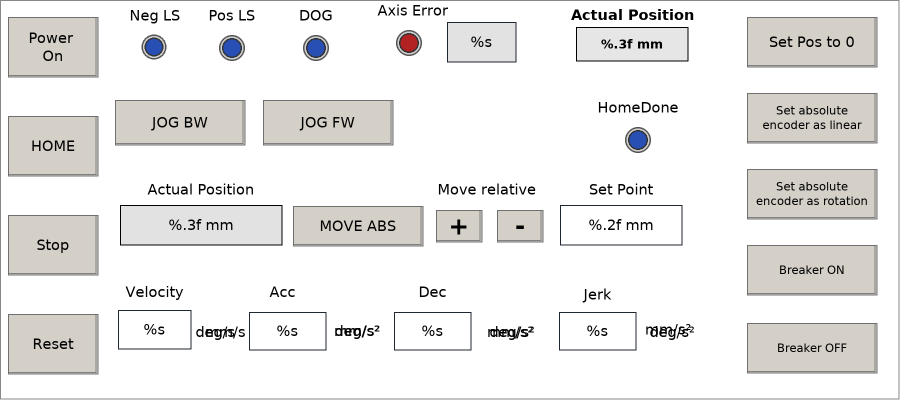
VISUALIZATION AxisHMI_Ex  // 900x400
VAR_IN_OUT
	stAxisHMI	: ST_MotionAxis_MC	;
	mcAxis		: FB_MotionAxis_MC;
	//sAxisName	: STRING			;// Axis Name
	//iAxisID		: INT			;// Axis Id
	xError		: BOOL				;// Axis error flag
END_VAR
    Button (115,100 130x45), "JOG BW", colour toggle: stAxisHMI.mcJog.JogBackwards
        OnMouseDown: execute { stAxisHMI.mcJog.JogBackwards := TRUE; }
        OnMouseUp: execute { stAxisHMI.mcJog.JogBackwards := FALSE; }
    Button (263,100 130x45), "JOG FW", colour toggle: stAxisHMI.mcJog.JogForward
        OnMouseDown: execute { stAxisHMI.mcJog.JogForward := TRUE; }
        OnMouseUp: execute { stAxisHMI.mcJog.JogForward := FALSE; }
    Rectangle (120,205 162x40), "%.3f mm", text variable: stAxisHMI.rActualPosHMI
        OnMouseClick: write the text variable via Default
    Label (141,177 120x25), "Actual Position"
    Button (8,17 90x60), "Power On", colour toggle: stAxisHMI.mcPower.Enable, pressed state: stAxisHMI.mcPower.Enable
        OnMouseClick: toggle stAxisHMI.mcPower.Enable
    Button (8,215 90x60), "Stop", colour toggle: stAxisHMI.mcStop.Execute, invisible if: NOT stAxisHMI.bStopButtonShow
        OnMouseDown: execute { stAxisHMI.mcStop.Execute := TRUE; }
        OnMouseUp: execute { stAxisHMI.mcStop.Execute := FALSE; }
    Button (8,314 90x60), "Reset", colour toggle: stAxisHMI.mcReset.Execute
        OnMouseDown: execute { stAxisHMI.mcReset.Execute := TRUE; }
        OnMouseUp: execute { stAxisHMI.mcReset.Execute := FALSE; }
    Label (111,277 87x30), "Velocity"
    Rectangle (118,310 73x39), "%s", text variable: stAxisHMI.rVeloPers
        OnMouseClick: write the text variable via Default, min 1, max stAxisHMI.rMaxVelocity
    Label (230,277 105x30), "Acc"
    Rectangle (249,312 77x38), "%s", text variable: stAxisHMI.rAcceleration
        OnMouseClick: write stAxisHMI.rAccPers via Default, min 1, max stAxisHMI.rMaxAcceleration
    Lamp1 (139,33 30x28), variable: stAxisHMI.bNegSen, invisible if: NOT stAxisHMI.bNegSensorShow, style: Lamp-Lamp1-Blue
    Label (364,-2 102x25), "Axis Error"
    Rectangle (447,22 69x40), "%s", text variable: stAxisHMI.mcReadStatus.ErrorID
    Lamp1 (394,28 30x30), variable: xError, style: Lamp-Lamp1-Red
    Lamp1 (217,33 30x30), variable: stAxisHMI.bPosSen, invisible if: NOT stAxisHMI.bPosSensorShow, style: Lamp-Lamp1-Blue
    Label (188,3 88x25), "Pos LS", invisible if: NOT stAxisHMI.bPosSensorShow
    Label (111,3 88x25), "Neg LS", invisible if: NOT stAxisHMI.bNegSensorShow
    Rectangle (560,205 122x40), "%.2f mm", text variable: stAxisHMI.rDistance
        OnMouseClick: write the text variable via Default, min 0, max stAxisHMI.rMaxDistance
    Button (293,206 130x40), "MOVE ABS", colour toggle: stAxisHMI.mcMoveAbsolute.Busy, pressed state: stAxisHMI.mcMoveAbsolute.Busy
        OnMouseDown: execute { stAxisHMI.bMoveAbsHMI := TRUE; }
        OnMouseUp: execute { stAxisHMI.bMoveAbsHMI := FALSE; }
    Label (561,177 120x25), "Set Point"
    Button (436,210 46x32), "+", colour toggle: stAxisHMI.mcMoveRelative.Busy, pressed state: stAxisHMI.mcMoveRelative.Busy
        OnMouseDown: execute { stAxisHMI.rPosition := stAxisHMI.rDistance; stAxisHMI.mcMoveRelative.Execute := TRUE; }
        OnMouseUp: execute { stAxisHMI.mcMoveRelative.Execute := FALSE; }
    Button (497,210 46x32), "-", colour toggle: stAxisHMI.mcMoveRelative.Busy, pressed state: stAxisHMI.mcMoveRelative.Busy
        OnMouseDown: execute { stAxisHMI.rPosition := -(stAxisHMI.rDistance); stAxisHMI.mcMoveRelative.Execute := TRUE; }
        OnMouseUp: execute { stAxisHMI.mcMoveRelative.Execute := FALSE; }
    Label (427,177 120x25), "Move relative"
    Label (330,316 55x30), "mm/s²"
    Label (196,317 59x30), "mm/s"
    Label (191,317 49x30), "deg/s", invisible if: NOT stAxisHMI.bUnitDegShow
    Label (328,316 59x30), "deg/s²", invisible if: NOT stAxisHMI.bUnitDegShow
    Label (380,277 105x30), "Dec"
    Rectangle (394,312 77x38), "%s", text variable: stAxisHMI.rDeceleration
        OnMouseClick: write stAxisHMI.rDecPers via Default, min 1, max stAxisHMI.rMaxDeceleration
    Label (483,317 55x30), "mm/s²"
    Label (483,317 59x30), "deg/s²", invisible if: NOT stAxisHMI.bUnitDegShow
    Button (8,116 90x60), "HOME", colour toggle: stAxisHMI.mcHome.Busy
        OnMouseDown: execute { mcAxis.mcHomeAxis.xExecute	:= TRUE; }
        OnMouseUp: execute { mcAxis.mcHomeAxis.xExecute	:= FALSE; }
    Rectangle (559,312 77x38), "%s", text variable: stAxisHMI.rJerk, invisible if: NOT stAxisHMI.bJerkShow
        OnMouseClick: write the text variable via Default, min 0, max stAxisHMI.rMaxJerk
    Label (572,282 51x25), "Jerk", invisible if: NOT stAxisHMI.bJerkShow
    Label (643,317 59x30), "deg/s²", invisible if: NOT stAxisHMI.bUnitDegShow
    Label (641,317 55x25), "mm/s²", invisible if: NOT stAxisHMI.bJerkShow
    Label (557,0 152x30), "Actual Position"
    Rectangle (576,27 112x34), "%.3f mm", text variable: stAxisHMI.rActualPos
    Lamp1 (301,33 30x30), variable: stAxisHMI.bPositionSensor, style: Lamp-Lamp1-Blue
    Label (272,3 88x25), "DOG", invisible if: NOT stAxisHMI.bPosSensorShow
    Lamp1 (623,125 30x30), variable: stAxisHMI.xHomingDone, style: Lamp-Lamp1-Blue
    Label (594,95 88x25), "HomeDone", invisible if: NOT stAxisHMI.bPosSensorShow
    Button (747,17 130x50), "Set Pos to 0", colour toggle: stAxisHMI.CoeWrt.bExecute
        OnMouseDown: execute {
            (*stAxisHMI.CoeWrt.bExecute := TRUE;
            stAxisHMI.nIndex	:= 16#2005;
            stAxisHMI.nSubIndex	:= 16#1F;
            stAxisHMI.iSdoWrite	:= 6;//clear encoder and set current position as origin*)
            stAxisHMI.mcPower.Enable	:= FALSE;
        }
        OnMouseUp: execute { stAxisHMI.iCoeWrt	:= 1; }
    Button (747,93 130x50), "Set absolute encoder as linear", colour toggle: stAxisHMI.CoeWrt.bExecute
        OnMouseDown: execute {
            (*stAxisHMI.CoeWrt.bExecute := TRUE;
            stAxisHMI.nIndex	:= 16#2002;
            stAxisHMI.nSubIndex	:= 16#02;
            stAxisHMI.iSdoWrite	:= 1;//linear mode*)
        }
        OnMouseUp: execute { (*stAxisHMI.CoeWrt.bExecute := FALSE;*) stAxisHMI.iCoeWrt	:= 2; }
    Button (747,169 130x50), "Set absolute encoder as rotation", colour toggle: stAxisHMI.CoeWrt.bExecute
        OnMouseDown: execute {
            (*stAxisHMI.CoeWrt.bExecute := TRUE;
            stAxisHMI.nIndex	:= 16#2002;
            stAxisHMI.nSubIndex	:= 16#02;
            stAxisHMI.iSdoWrite	:= 2;//rotate mode*)
        }
        OnMouseUp: execute { (*stAxisHMI.CoeWrt.bExecute := FALSE;*) stAxisHMI.iCoeWrt	:= 3; }
    Button (747,245 130x50), "Breaker ON", colour toggle: stAxisHMI.CoeWrt.bExecute
        OnMouseDown: execute {
            (*stAxisHMI.CoeWrt.bExecute := TRUE;
            stAxisHMI.nIndex	:= 16#2004;
            stAxisHMI.nSubIndex	:= 16#06;
            stAxisHMI.iSdoWrite	:= 1;//rotate mode*)
        }
        OnMouseUp: execute { (*stAxisHMI.CoeWrt.bExecute := FALSE;*) stAxisHMI.iCoeWrt	:= 4; }
    Button (747,323 130x50), "Breaker OFF", colour toggle: stAxisHMI.CoeWrt.bExecute
        OnMouseDown: execute {
            (*stAxisHMI.CoeWrt.bExecute := TRUE;
            stAxisHMI.nIndex	:= 16#2004;
            stAxisHMI.nSubIndex	:= 16#06;
            stAxisHMI.iSdoWrite	:= 0;//*)
        }
        OnMouseUp: execute { (*stAxisHMI.CoeWrt.bExecute := FALSE;*) stAxisHMI.iCoeWrt	:= 5; }
END_VISUALIZATION

(* stored: Version 1.1.0.1, ProductVersion 3.1.4024.12
   Visu AxisHMI_Ex: Id {ea0d0bd1-41cf-46ee-9787-e31362f65919} *)
